Fanuc KAREL source: kb00063.KL

-- PROVISIONAL review KL for V770-1; original PC SHA256 a3b9bca23bea72a1b46f67f5704bedc6c4eabbbcd40b146c8c4917924cfdde4a
-- Incomplete behavior may be omitted. Consult companion uncertainty JSON. Do not deploy.
PROGRAM KB00063
%NOLOCKGROUP
BEGIN
  -- UNRESOLVED_PC offsets 5-12; opcodes 9D,23
  -- UNRESOLVED_PC offsets 17-24; opcodes 9D,23
  -- UNRESOLVED_PC offsets 29-36; opcodes 9D,23
  -- UNRESOLVED_PC offsets 41-63; opcodes 27,22,22,22,31
  -- UNRESOLVED_PC offsets 68-72; opcodes 7F
END KB00063
